// TIA Portal V16 export
// export: Created 2022-01-12T14:34:27.6170037Z, ExportSetting WithDefaults, DisplayName Totally Integrated Automation Portal, DisplayVersion V16 Update 4, DisplayName TIA Portal Version Control Interface, DisplayVersion V16 Update 2, DisplayName TIA Portal Openness, DisplayVersion V16 Update 4, DisplayName STEP 7 Professional, DisplayVersion V16 Update 4, DisplayName STEP 7 Safety, DisplayVersion V16, DisplayName WinCC Professional, DisplayVersion V16 Update 4
TYPE "typSetReset"
// stored: IsFailsafeCompliant false
   STRUCT
      inSet : Bool;
      inReset : Bool;
      czasDoSet : Int;
      czasDoReset : Int;
      wyjście : Bool;
      setCzas : Int;
      resetCzas : Int;
   END_STRUCT;
END_TYPE
